{attribute 'qualified_only'}
TYPE E_ApproachDirection :
(
	Positive_X := 0,
	Positive_Y := 1,
	Positive_Z := 2,
	Negative_X := 3,
	Negative_Y := 4,
	Negative_Z := 5
);
END_TYPE

(* stored: Version 1.1.0.1
   DUT E_ApproachDirection: Id {382155ab-2f44-479a-9a93-f3a4e6426391} *)
